(* IEC 61131-3 sources: s22-soft-shell/ST_resources/examples, 8 files *)

(* ---- expression_add.st ---- *)
PROGRAM expression_add
VAR
    a: int;
END_VAR
a := (1 + 2)
END_PROGRAM

(* ---- expression_add_mul.st ---- *)
PROGRAM expression_add_mul
VAR
    a: int;
END_VAR
a := (2 + 4) * (1 + 3);
END_PROGRAM

(* ---- expression_div.st ---- *)
PROGRAM expression_div
VAR
    a: int;
END_VAR
a := (10 / 2)
END_PROGRAM

(* ---- expression_mul.st ---- *)
PROGRAM expression_mul
VAR
    a: int;
END_VAR
a := (3 * 2)
END_PROGRAM

(* ---- IF_1.st ---- *)
PROGRAM IF_1
    VAR
        x : INT
        y : BOOL;
    END_VAR
    x :=2
    IF x = 2 THEN
        x := 3
END_PROGRAM

(* ---- simple_1.st ---- *)
PROGRAM simple_1
    VAR
		a : INT;
    END_VAR
		a := 1;
END_PROGRAM

(* ---- simple_2.st ---- *)
PROGRAM simple_2
    VAR
		a : real;
    END_VAR
		a := 1.2;
END_PROGRAM

(* ---- simple_3.st ---- *)
PROGRAM simple_3
    VAR
		a : real;
        b : int
    END_VAR
		a := 1.2;
        b := a;
END_PROGRAM
